% RSLogix 500 project 2 Head Filler - Reautomation.RSS, saved by version 7.00.00.19 %
PROJECT "ACINEW07"    % processor: MicroLogix 1200 %

PROGRAM FILES
  LAD 2 "MAIN"  15 rungs
  LAD 3 "FILL SEQ"  10 rungs
  LAD 4 "RESET"  12 rungs
  LAD 5 "HMI"  10 rungs
  LAD 6 "RECAP"  12 rungs

DATA FILES
  O0 OUTPUT  4 elements
  I1 INPUT  4 elements
  S2 STATUS  66 elements
  B3 BINARY  21 elements
  T4 TIMER  38 elements
  C5 COUNTER  1 elements
  R6 CONTROL  1 elements
  N7 INTEGER  7 elements
  F8 FLOAT  1 elements
  L9   1 elements

LADDER 2 "MAIN"
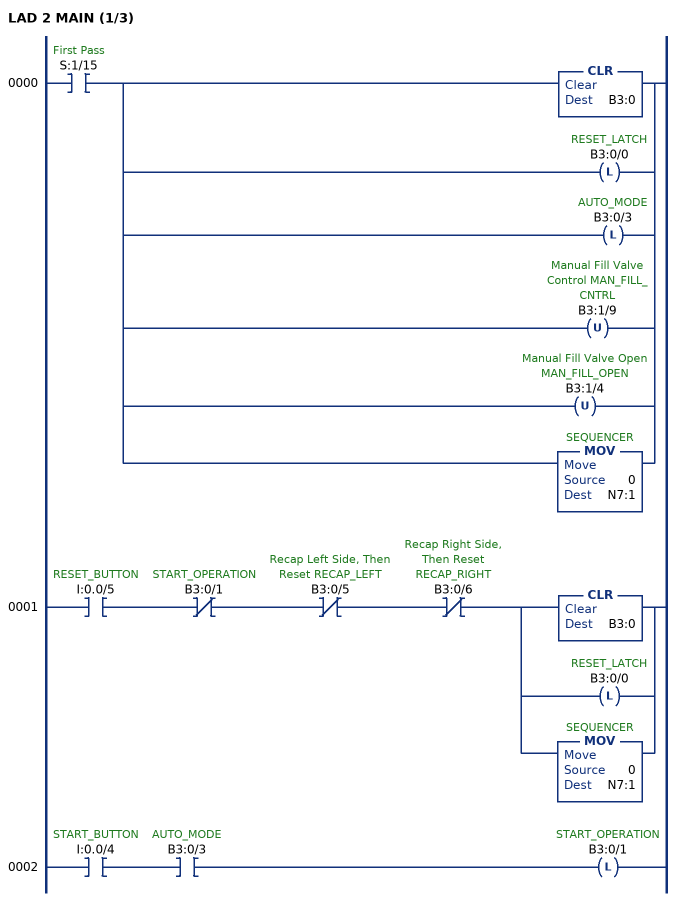
% Rung: 0 %
SOR XIC S:1/15 BST CLR B3:0 NXB OTL B3:0/0 NXB OTL B3:0/3 NXB OTU B3:1/9 NXB OTU B3:1/4 NXB MOV 0 N7:1 BND EOR
%   S:1/15  "First Pass" %
%   B3:0/0  RESET_LATCH %
%   B3:0/3  AUTO_MODE %
%   B3:1/9  MAN_FILL_CNTRL  "Manual Fill Valve Control" %
%   B3:1/4  MAN_FILL_OPEN  "Manual Fill Valve Open" %
%   N7:1  SEQUENCER %
% Rung: 1 %
SOR XIC I:0.0/5 XIO B3:0/1 XIO B3:0/5 XIO B3:0/6 BST CLR B3:0 NXB OTL B3:0/0 NXB MOV 0 N7:1 BND EOR
%   I:0.0/5  RESET_BUTTON %
%   B3:0/1  START_OPERATION %
%   B3:0/5  RECAP_LEFT  "Recap Left Side, Then Reset" %
%   B3:0/6  RECAP_RIGHT  "Recap Right Side, Then Reset" %
%   B3:0/0  RESET_LATCH %
%   N7:1  SEQUENCER %
% Rung: 2 %
SOR XIC I:0.0/4 XIC B3:0/3 OTL B3:0/1 EOR
%   I:0.0/4  START_BUTTON %
%   B3:0/3  AUTO_MODE %
%   B3:0/1  START_OPERATION %

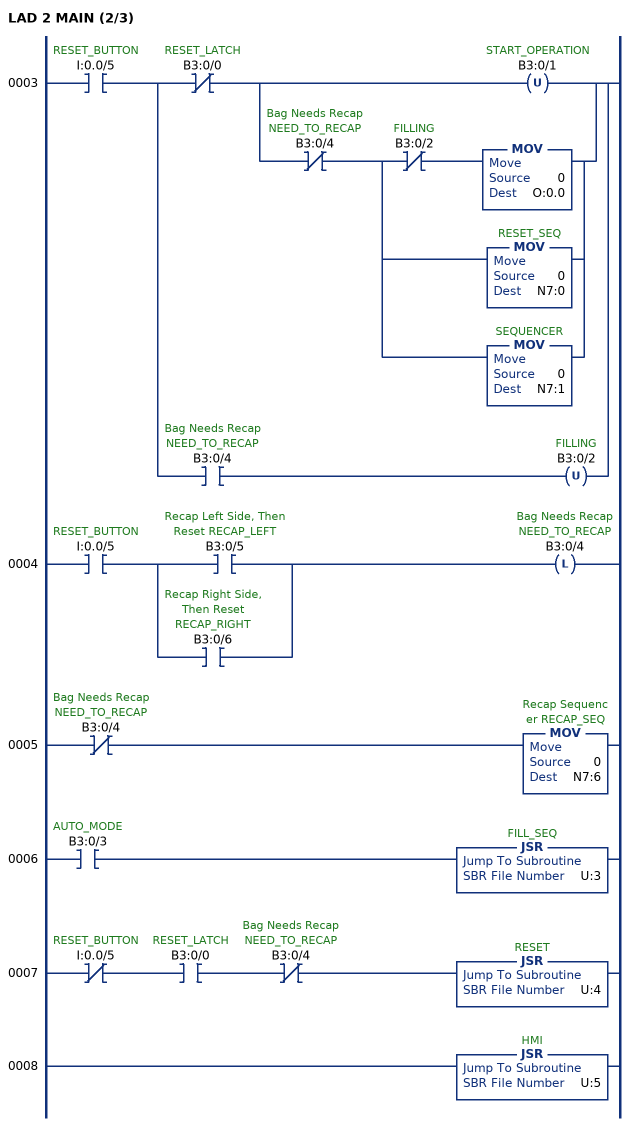
% Rung: 3 %
SOR XIC I:0.0/5 BST XIO B3:0/0 BST OTU B3:0/1 NXB XIO B3:0/4 BST XIO B3:0/2 MOV 0 O:0.0 NXB MOV 0 N7:0 NXB MOV 0 N7:1 BND BND NXB XIC B3:0/4 OTU B3:0/2 BND EOR
%   I:0.0/5  RESET_BUTTON %
%   B3:0/0  RESET_LATCH %
%   B3:0/1  START_OPERATION %
%   B3:0/4  NEED_TO_RECAP  "Bag Needs Recap" %
%   B3:0/2  FILLING %
%   N7:0  RESET_SEQ %
%   N7:1  SEQUENCER %
% Rung: 4 %
SOR XIC I:0.0/5 BST XIC B3:0/5 NXB XIC B3:0/6 BND OTL B3:0/4 EOR
%   I:0.0/5  RESET_BUTTON %
%   B3:0/5  RECAP_LEFT  "Recap Left Side, Then Reset" %
%   B3:0/6  RECAP_RIGHT  "Recap Right Side, Then Reset" %
%   B3:0/4  NEED_TO_RECAP  "Bag Needs Recap" %
% Rung: 5 %
SOR XIO B3:0/4 MOV 0 N7:6 EOR
%   B3:0/4  NEED_TO_RECAP  "Bag Needs Recap" %
%   N7:6  RECAP_SEQ  "Recap Sequencer" %
% Rung: 6 %
SOR XIC B3:0/3 JSR U:3 EOR
%   B3:0/3  AUTO_MODE %
%   U:3  FILL_SEQ %
% Rung: 7 %
SOR XIO I:0.0/5 XIC B3:0/0 XIO B3:0/4 JSR U:4 EOR
%   I:0.0/5  RESET_BUTTON %
%   B3:0/0  RESET_LATCH %
%   B3:0/4  NEED_TO_RECAP  "Bag Needs Recap" %
%   U:4  RESET %
% Rung: 8 %
SOR JSR U:5 EOR
%   U:5  HMI %

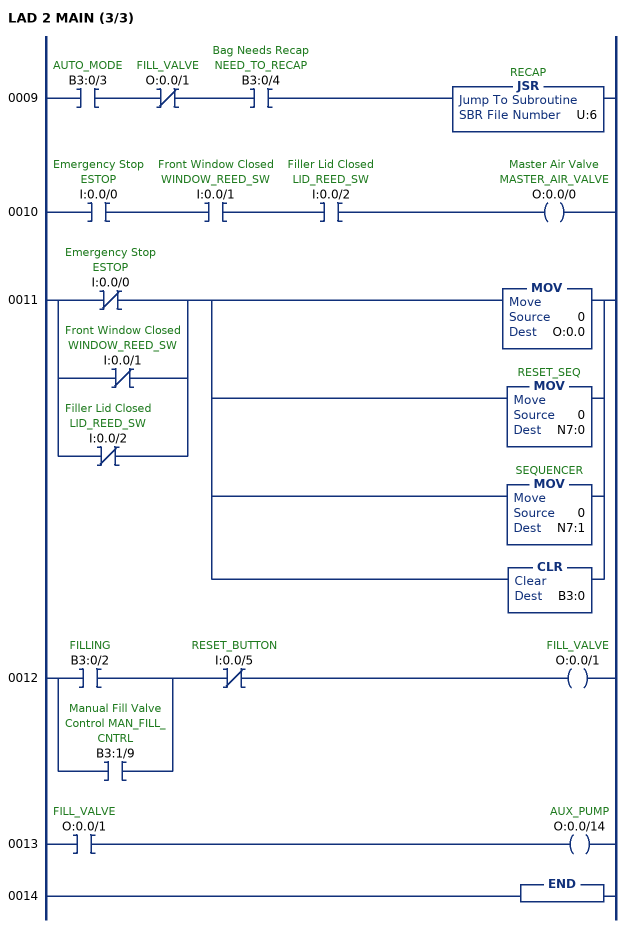
% Rung: 9 %
SOR XIC B3:0/3 XIO O:0.0/1 XIC B3:0/4 JSR U:6 EOR
%   B3:0/3  AUTO_MODE %
%   O:0.0/1  FILL_VALVE %
%   B3:0/4  NEED_TO_RECAP  "Bag Needs Recap" %
%   U:6  RECAP %
% Rung: 10 %
SOR XIC I:0.0/0 XIC I:0.0/1 XIC I:0.0/2 OTE O:0.0/0 EOR
%   I:0.0/0  ESTOP  "Emergency Stop" %
%   I:0.0/1  WINDOW_REED_SW  "Front Window Closed" %
%   I:0.0/2  LID_REED_SW  "Filler Lid Closed" %
%   O:0.0/0  MASTER_AIR_VALVE  "Master Air Valve" %
% Rung: 11 %
SOR BST XIO I:0.0/0 NXB XIO I:0.0/1 NXB XIO I:0.0/2 BND BST MOV 0 O:0.0 NXB MOV 0 N7:0 NXB MOV 0 N7:1 NXB CLR B3:0 BND EOR
%   I:0.0/0  ESTOP  "Emergency Stop" %
%   I:0.0/1  WINDOW_REED_SW  "Front Window Closed" %
%   I:0.0/2  LID_REED_SW  "Filler Lid Closed" %
%   N7:0  RESET_SEQ %
%   N7:1  SEQUENCER %
% Rung: 12 %
SOR BST XIC B3:0/2 NXB XIC B3:1/9 BND XIO I:0.0/5 OTE O:0.0/1 EOR
%   B3:0/2  FILLING %
%   B3:1/9  MAN_FILL_CNTRL  "Manual Fill Valve Control" %
%   I:0.0/5  RESET_BUTTON %
%   O:0.0/1  FILL_VALVE %
% Rung: 13 %
SOR XIC O:0.0/1 OTE O:0.0/14 EOR
%   O:0.0/1  FILL_VALVE %
%   O:0.0/14  AUX_PUMP %
% Rung: 14 %
SOR END EOR

LADDER 3 "FILL SEQ"
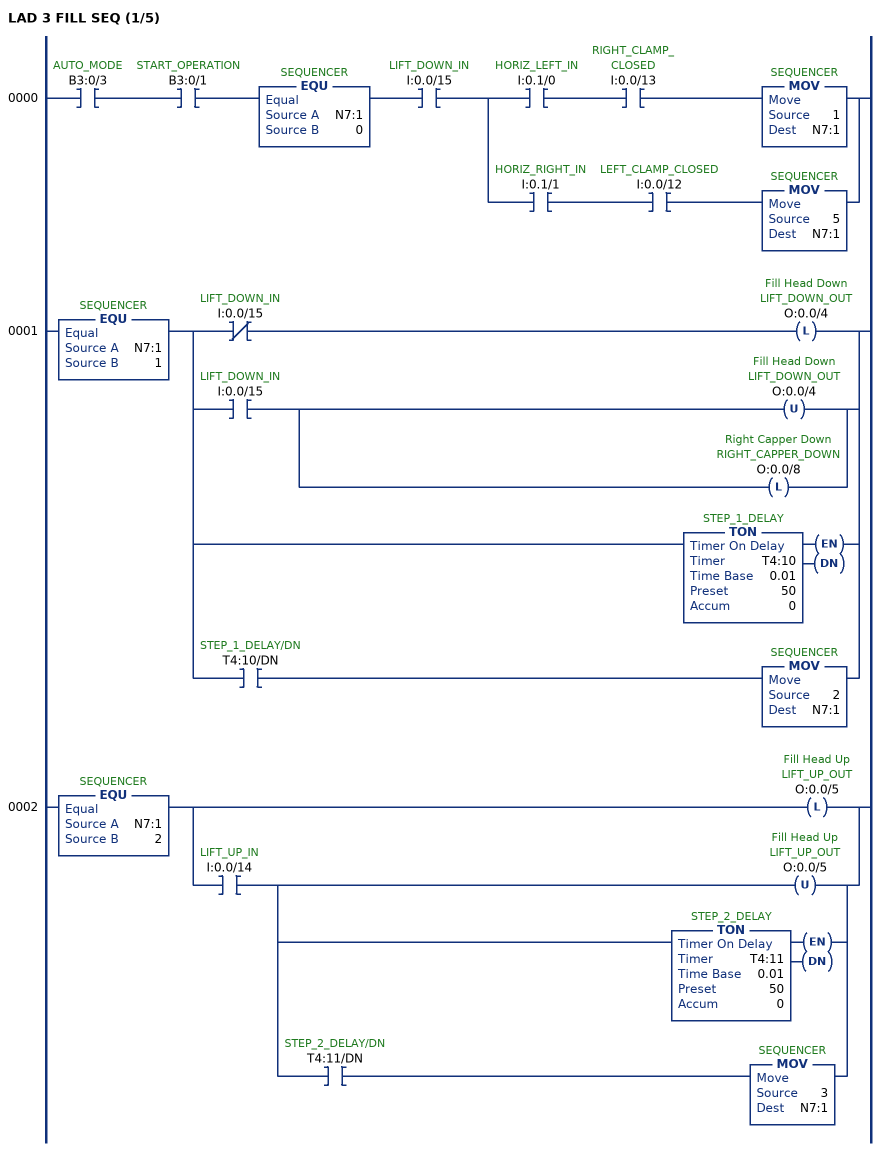
% Rung: 0 %
SOR XIC B3:0/3 XIC B3:0/1 EQU N7:1 0 XIC I:0.0/15 BST XIC I:0.1/0 XIC I:0.0/13 MOV 1 N7:1 NXB XIC I:0.1/1 XIC I:0.0/12 MOV 5 N7:1 BND EOR
%   B3:0/3  AUTO_MODE %
%   B3:0/1  START_OPERATION %
%   N7:1  SEQUENCER %
%   I:0.0/15  LIFT_DOWN_IN %
%   I:0.1/0  HORIZ_LEFT_IN %
%   I:0.0/13  RIGHT_CLAMP_CLOSED %
%   I:0.1/1  HORIZ_RIGHT_IN %
%   I:0.0/12  LEFT_CLAMP_CLOSED %
% Rung: 1 %
SOR EQU N7:1 1 BST XIO I:0.0/15 OTL O:0.0/4 NXB XIC I:0.0/15 BST OTU O:0.0/4 NXB OTL O:0.0/8 BND NXB TON T4:10 0.01 50 0 NXB XIC T4:10/DN MOV 2 N7:1 BND EOR
%   N7:1  SEQUENCER %
%   I:0.0/15  LIFT_DOWN_IN %
%   O:0.0/4  LIFT_DOWN_OUT  "Fill Head Down" %
%   O:0.0/8  RIGHT_CAPPER_DOWN  "Right Capper Down" %
%   T4:10  STEP_1_DELAY %
% Rung: 2 %
SOR EQU N7:1 2 BST OTL O:0.0/5 NXB XIC I:0.0/14 BST OTU O:0.0/5 NXB TON T4:11 0.01 50 0 NXB XIC T4:11/DN MOV 3 N7:1 BND BND EOR
%   N7:1  SEQUENCER %
%   O:0.0/5  LIFT_UP_OUT  "Fill Head Up" %
%   I:0.0/14  LIFT_UP_IN %
%   T4:11  STEP_2_DELAY %

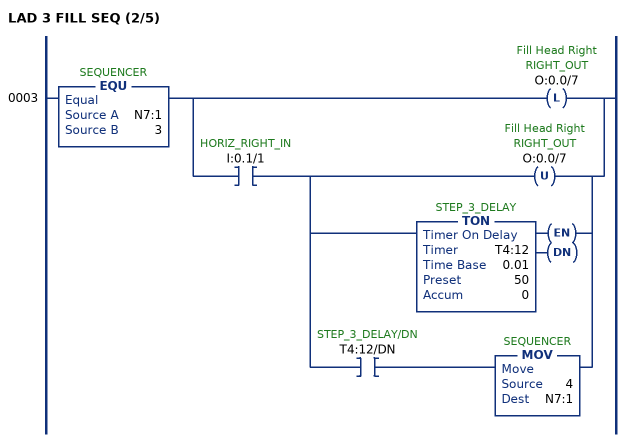
% Rung: 3 %
SOR EQU N7:1 3 BST OTL O:0.0/7 NXB XIC I:0.1/1 BST OTU O:0.0/7 NXB TON T4:12 0.01 50 0 NXB XIC T4:12/DN MOV 4 N7:1 BND BND EOR
%   N7:1  SEQUENCER %
%   O:0.0/7  RIGHT_OUT  "Fill Head Right" %
%   I:0.1/1  HORIZ_RIGHT_IN %
%   T4:12  STEP_3_DELAY %

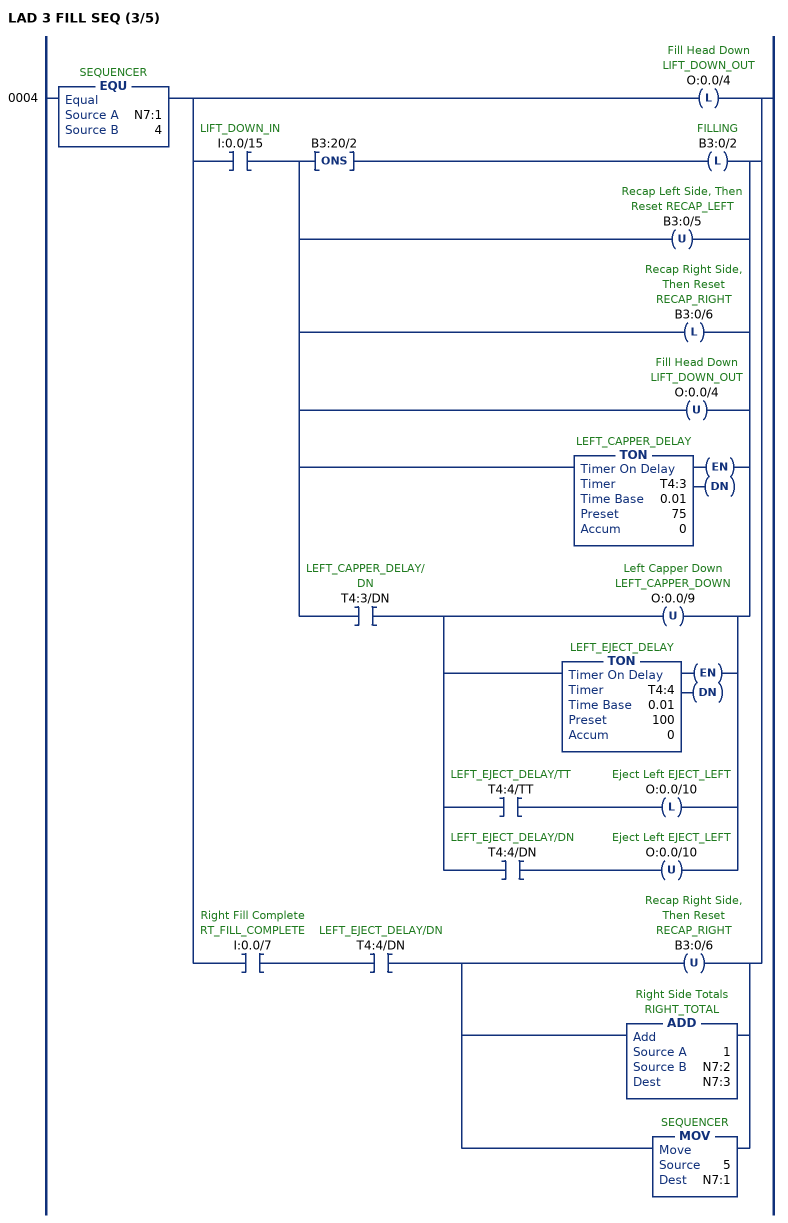
% Rung: 4 %
SOR EQU N7:1 4 BST OTL O:0.0/4 NXB XIC I:0.0/15 BST ONS B3:20/2 OTL B3:0/2 NXB OTU B3:0/5 NXB OTL B3:0/6 NXB OTU O:0.0/4 NXB TON T4:3 0.01 75 0 NXB XIC T4:3/DN BST OTU O:0.0/9 NXB TON T4:4 0.01 100 0 NXB XIC T4:4/TT OTL O:0.0/10 NXB XIC T4:4/DN OTU O:0.0/10 BND BND NXB XIC I:0.0/7 XIC T4:4/DN BST OTU B3:0/6 NXB ADD 1 N7:2 N7:3 NXB MOV 5 N7:1 BND BND EOR
%   N7:1  SEQUENCER %
%   O:0.0/4  LIFT_DOWN_OUT  "Fill Head Down" %
%   I:0.0/15  LIFT_DOWN_IN %
%   B3:0/2  FILLING %
%   B3:0/5  RECAP_LEFT  "Recap Left Side, Then Reset" %
%   B3:0/6  RECAP_RIGHT  "Recap Right Side, Then Reset" %
%   T4:3  LEFT_CAPPER_DELAY %
%   O:0.0/9  LEFT_CAPPER_DOWN  "Left Capper Down" %
%   T4:4  LEFT_EJECT_DELAY %
%   O:0.0/10  EJECT_LEFT  "Eject Left" %
%   I:0.0/7  RT_FILL_COMPLETE  "Right Fill Complete" %
%   N7:2  LEFT_TOTAL  "Left Side Totals" %
%   N7:3  RIGHT_TOTAL  "Right Side Totals" %

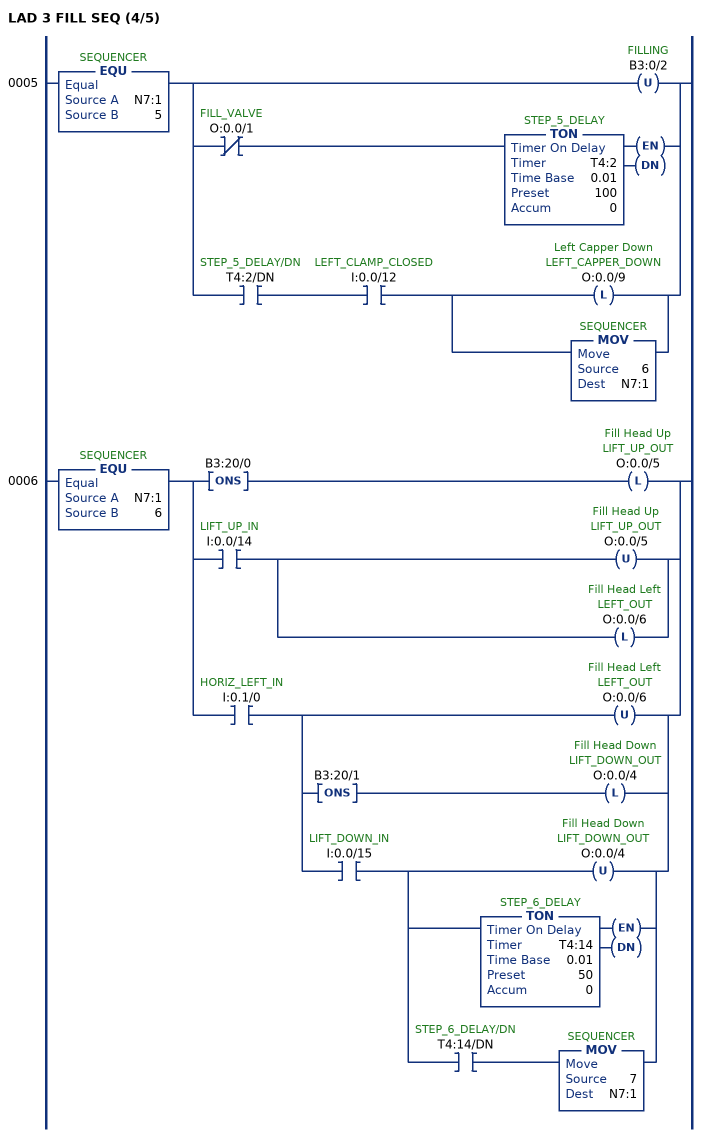
% Rung: 5 %
SOR EQU N7:1 5 BST OTU B3:0/2 NXB XIO O:0.0/1 TON T4:2 0.01 100 0 NXB XIC T4:2/DN XIC I:0.0/12 BST OTL O:0.0/9 NXB MOV 6 N7:1 BND BND EOR
%   N7:1  SEQUENCER %
%   B3:0/2  FILLING %
%   O:0.0/1  FILL_VALVE %
%   T4:2  STEP_5_DELAY %
%   I:0.0/12  LEFT_CLAMP_CLOSED %
%   O:0.0/9  LEFT_CAPPER_DOWN  "Left Capper Down" %
% Rung: 6 %
SOR EQU N7:1 6 BST ONS B3:20/0 OTL O:0.0/5 NXB BST XIC I:0.0/14 BST OTU O:0.0/5 NXB OTL O:0.0/6 BND NXB XIC I:0.1/0 BST OTU O:0.0/6 NXB ONS B3:20/1 OTL O:0.0/4 NXB XIC I:0.0/15 BST OTU O:0.0/4 NXB TON T4:14 0.01 50 0 NXB XIC T4:14/DN MOV 7 N7:1 BND BND BND BND EOR
%   N7:1  SEQUENCER %
%   O:0.0/5  LIFT_UP_OUT  "Fill Head Up" %
%   I:0.0/14  LIFT_UP_IN %
%   O:0.0/6  LEFT_OUT  "Fill Head Left" %
%   I:0.1/0  HORIZ_LEFT_IN %
%   O:0.0/4  LIFT_DOWN_OUT  "Fill Head Down" %
%   I:0.0/15  LIFT_DOWN_IN %
%   T4:14  STEP_6_DELAY %

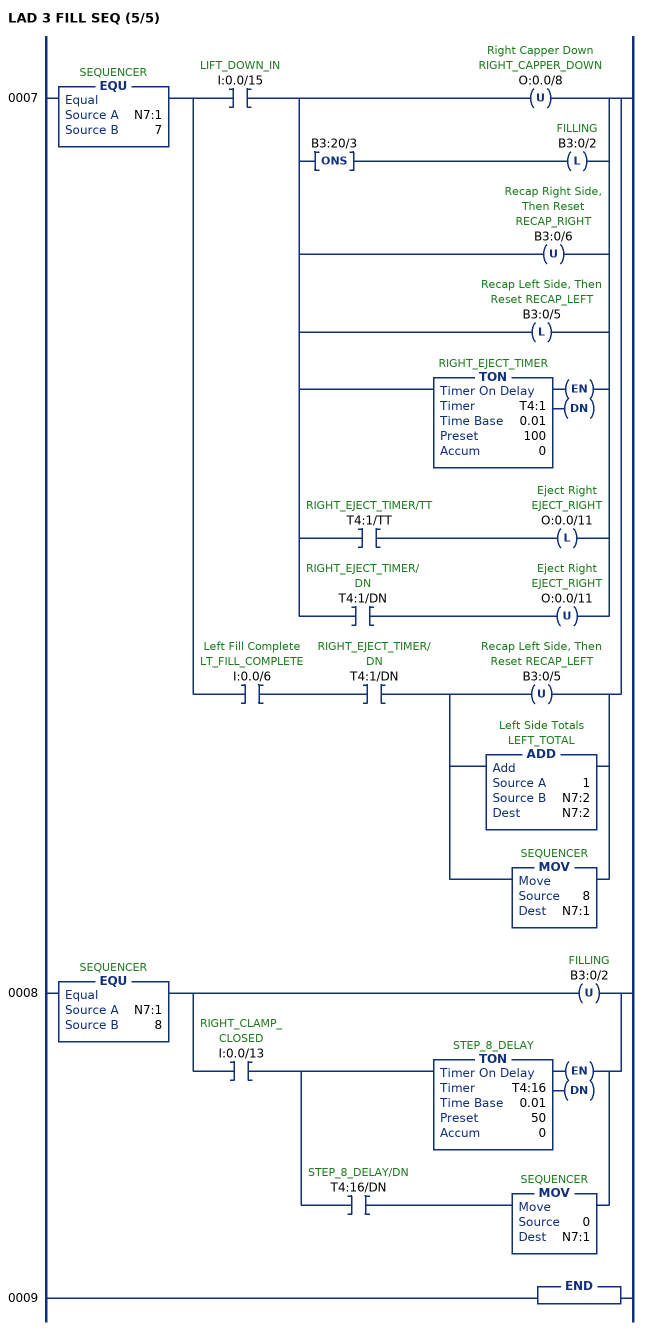
% Rung: 7 %
SOR EQU N7:1 7 BST XIC I:0.0/15 BST OTU O:0.0/8 NXB ONS B3:20/3 OTL B3:0/2 NXB OTU B3:0/6 NXB OTL B3:0/5 NXB TON T4:1 0.01 100 0 NXB XIC T4:1/TT OTL O:0.0/11 NXB XIC T4:1/DN OTU O:0.0/11 BND NXB XIC I:0.0/6 XIC T4:1/DN BST OTU B3:0/5 NXB ADD 1 N7:2 N7:2 NXB MOV 8 N7:1 BND BND EOR
%   N7:1  SEQUENCER %
%   I:0.0/15  LIFT_DOWN_IN %
%   O:0.0/8  RIGHT_CAPPER_DOWN  "Right Capper Down" %
%   B3:0/2  FILLING %
%   B3:0/6  RECAP_RIGHT  "Recap Right Side, Then Reset" %
%   B3:0/5  RECAP_LEFT  "Recap Left Side, Then Reset" %
%   T4:1  RIGHT_EJECT_TIMER %
%   O:0.0/11  EJECT_RIGHT  "Eject Right" %
%   I:0.0/6  LT_FILL_COMPLETE  "Left Fill Complete" %
%   N7:2  LEFT_TOTAL  "Left Side Totals" %
% Rung: 8 %
SOR EQU N7:1 8 BST OTU B3:0/2 NXB XIC I:0.0/13 BST TON T4:16 0.01 50 0 NXB XIC T4:16/DN MOV 0 N7:1 BND BND EOR
%   N7:1  SEQUENCER %
%   B3:0/2  FILLING %
%   I:0.0/13  RIGHT_CLAMP_CLOSED %
%   T4:16  STEP_8_DELAY %
% Rung: 9 %
SOR END EOR

LADDER 4 "RESET"
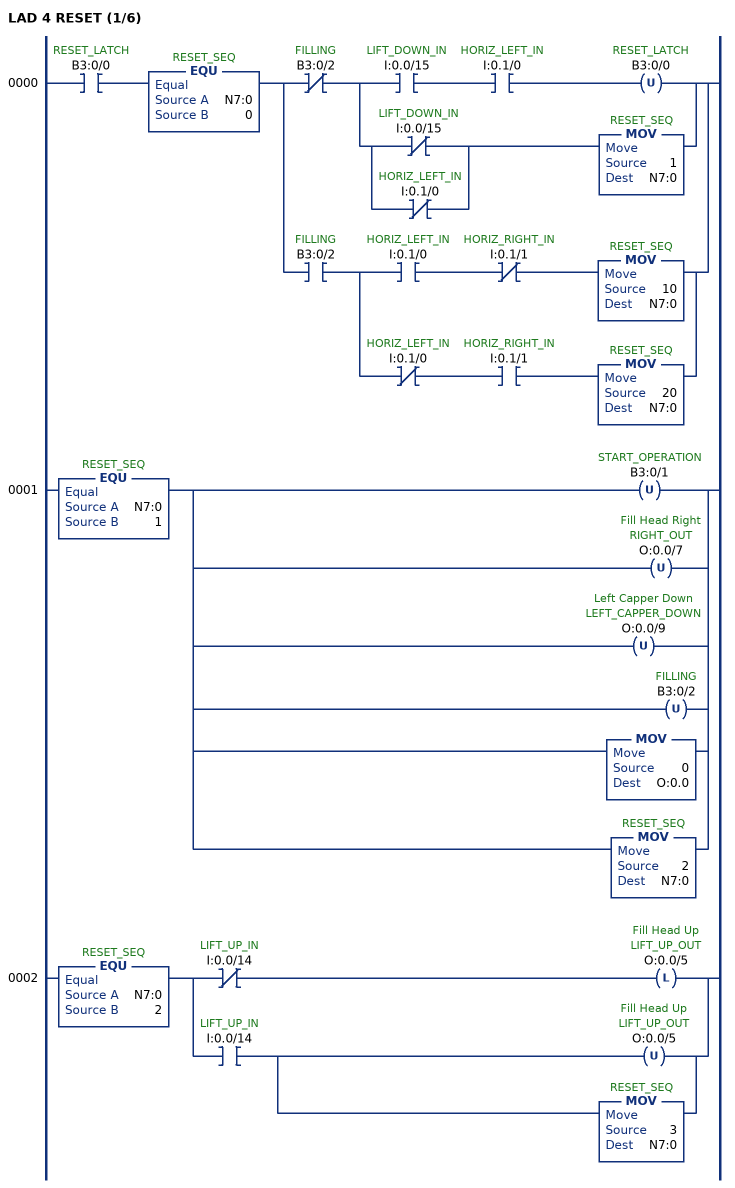
% Rung: 0 %
SOR XIC B3:0/0 EQU N7:0 0 BST XIO B3:0/2 BST XIC I:0.0/15 XIC I:0.1/0 OTU B3:0/0 NXB BST XIO I:0.0/15 NXB XIO I:0.1/0 BND MOV 1 N7:0 BND NXB XIC B3:0/2 BST XIC I:0.1/0 XIO I:0.1/1 MOV 10 N7:0 NXB XIO I:0.1/0 XIC I:0.1/1 MOV 20 N7:0 BND BND EOR
%   B3:0/0  RESET_LATCH %
%   N7:0  RESET_SEQ %
%   B3:0/2  FILLING %
%   I:0.0/15  LIFT_DOWN_IN %
%   I:0.1/0  HORIZ_LEFT_IN %
%   I:0.1/1  HORIZ_RIGHT_IN %
% Rung: 1 %
SOR EQU N7:0 1 BST OTU B3:0/1 NXB OTU O:0.0/7 NXB OTU O:0.0/9 NXB OTU B3:0/2 NXB MOV 0 O:0.0 NXB MOV 2 N7:0 BND EOR
%   N7:0  RESET_SEQ %
%   B3:0/1  START_OPERATION %
%   O:0.0/7  RIGHT_OUT  "Fill Head Right" %
%   O:0.0/9  LEFT_CAPPER_DOWN  "Left Capper Down" %
%   B3:0/2  FILLING %
% Rung: 2 %
SOR EQU N7:0 2 BST XIO I:0.0/14 OTL O:0.0/5 NXB XIC I:0.0/14 BST OTU O:0.0/5 NXB MOV 3 N7:0 BND BND EOR
%   N7:0  RESET_SEQ %
%   I:0.0/14  LIFT_UP_IN %
%   O:0.0/5  LIFT_UP_OUT  "Fill Head Up" %

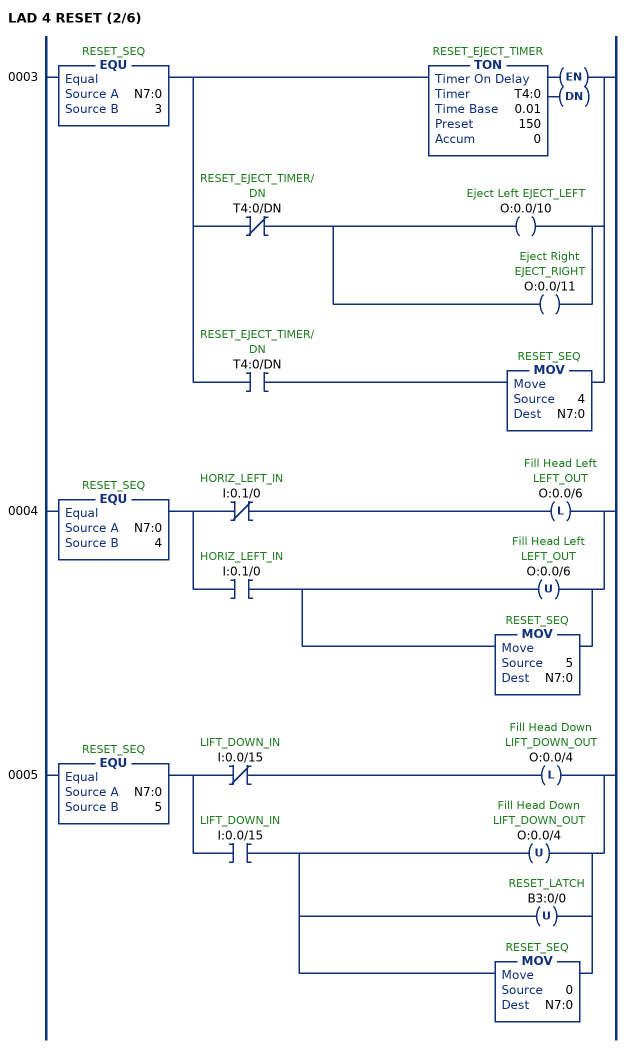
% Rung: 3 %
SOR EQU N7:0 3 BST TON T4:0 0.01 150 0 NXB XIO T4:0/DN BST OTE O:0.0/10 NXB OTE O:0.0/11 BND NXB XIC T4:0/DN MOV 4 N7:0 BND EOR
%   N7:0  RESET_SEQ %
%   T4:0  RESET_EJECT_TIMER %
%   O:0.0/10  EJECT_LEFT  "Eject Left" %
%   O:0.0/11  EJECT_RIGHT  "Eject Right" %
% Rung: 4 %
SOR EQU N7:0 4 BST XIO I:0.1/0 OTL O:0.0/6 NXB XIC I:0.1/0 BST OTU O:0.0/6 NXB MOV 5 N7:0 BND BND EOR
%   N7:0  RESET_SEQ %
%   I:0.1/0  HORIZ_LEFT_IN %
%   O:0.0/6  LEFT_OUT  "Fill Head Left" %
% Rung: 5 %
SOR EQU N7:0 5 BST XIO I:0.0/15 OTL O:0.0/4 NXB XIC I:0.0/15 BST OTU O:0.0/4 NXB OTU B3:0/0 NXB MOV 0 N7:0 BND BND EOR
%   N7:0  RESET_SEQ %
%   I:0.0/15  LIFT_DOWN_IN %
%   O:0.0/4  LIFT_DOWN_OUT  "Fill Head Down" %
%   B3:0/0  RESET_LATCH %

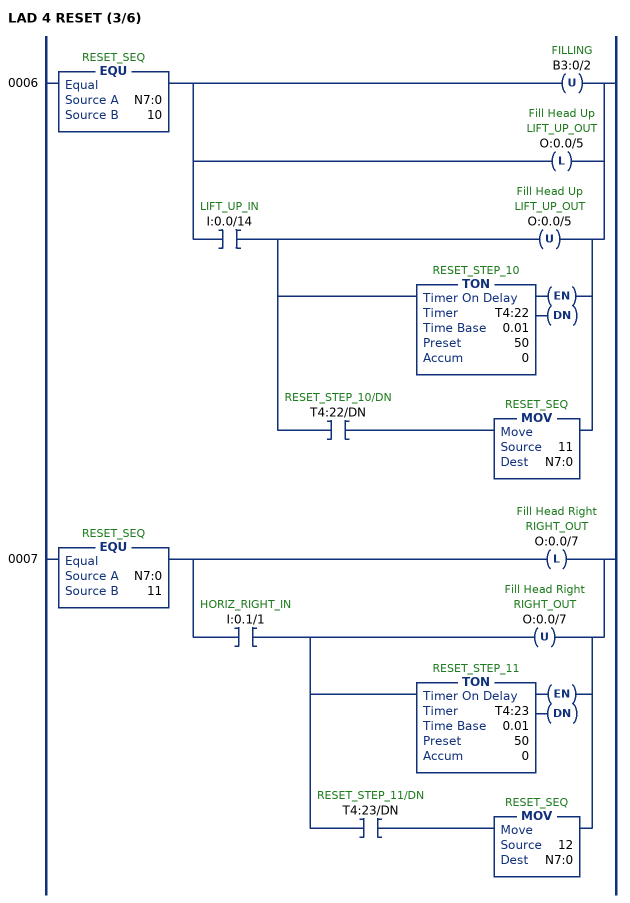
% Rung: 6 %
SOR EQU N7:0 10 BST OTU B3:0/2 NXB OTL O:0.0/5 NXB XIC I:0.0/14 BST OTU O:0.0/5 NXB TON T4:22 0.01 50 0 NXB XIC T4:22/DN MOV 11 N7:0 BND BND EOR
%   N7:0  RESET_SEQ %
%   B3:0/2  FILLING %
%   O:0.0/5  LIFT_UP_OUT  "Fill Head Up" %
%   I:0.0/14  LIFT_UP_IN %
%   T4:22  RESET_STEP_10 %
% Rung: 7 %
SOR EQU N7:0 11 BST OTL O:0.0/7 NXB XIC I:0.1/1 BST OTU O:0.0/7 NXB TON T4:23 0.01 50 0 NXB XIC T4:23/DN MOV 12 N7:0 BND BND EOR
%   N7:0  RESET_SEQ %
%   O:0.0/7  RIGHT_OUT  "Fill Head Right" %
%   I:0.1/1  HORIZ_RIGHT_IN %
%   T4:23  RESET_STEP_11 %

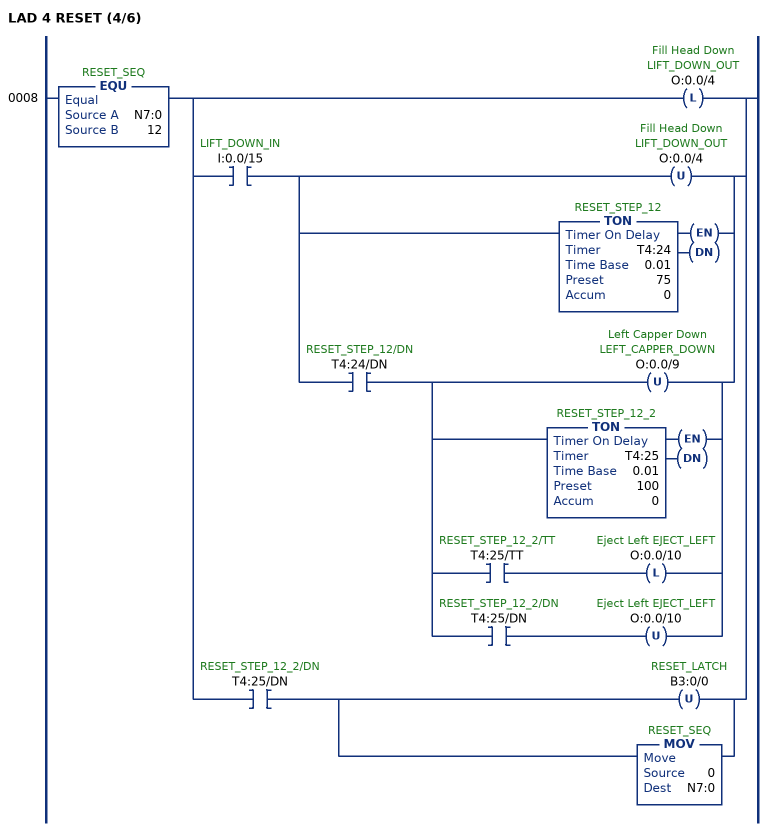
% Rung: 8 %
SOR EQU N7:0 12 BST OTL O:0.0/4 NXB XIC I:0.0/15 BST OTU O:0.0/4 NXB TON T4:24 0.01 75 0 NXB XIC T4:24/DN BST OTU O:0.0/9 NXB TON T4:25 0.01 100 0 NXB XIC T4:25/TT OTL O:0.0/10 NXB XIC T4:25/DN OTU O:0.0/10 BND BND NXB XIC T4:25/DN BST OTU B3:0/0 NXB MOV 0 N7:0 BND BND EOR
%   N7:0  RESET_SEQ %
%   O:0.0/4  LIFT_DOWN_OUT  "Fill Head Down" %
%   I:0.0/15  LIFT_DOWN_IN %
%   T4:24  RESET_STEP_12 %
%   O:0.0/9  LEFT_CAPPER_DOWN  "Left Capper Down" %
%   T4:25  RESET_STEP_12_2 %
%   O:0.0/10  EJECT_LEFT  "Eject Left" %
%   B3:0/0  RESET_LATCH %

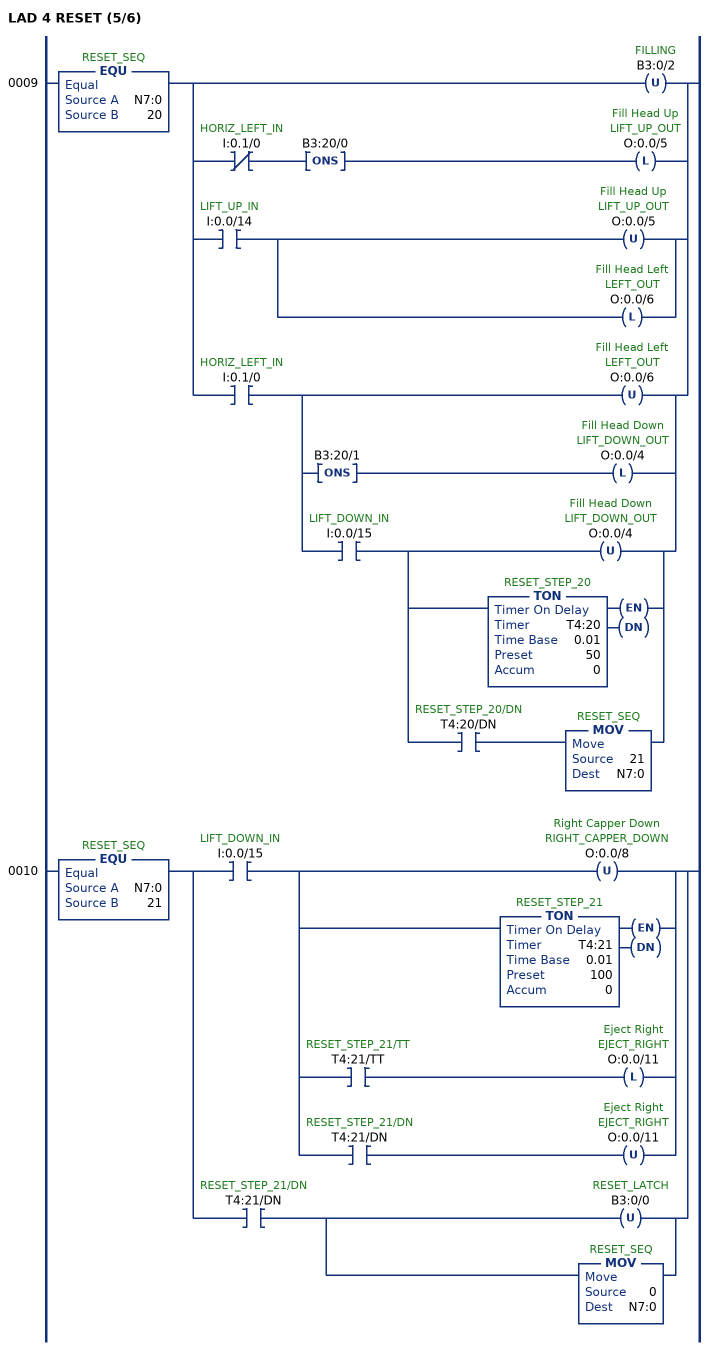
% Rung: 9 %
SOR EQU N7:0 20 BST OTU B3:0/2 NXB XIO I:0.1/0 ONS B3:20/0 OTL O:0.0/5 NXB BST XIC I:0.0/14 BST OTU O:0.0/5 NXB OTL O:0.0/6 BND NXB XIC I:0.1/0 BST OTU O:0.0/6 NXB ONS B3:20/1 OTL O:0.0/4 NXB XIC I:0.0/15 BST OTU O:0.0/4 NXB TON T4:20 0.01 50 0 NXB XIC T4:20/DN MOV 21 N7:0 BND BND BND BND EOR
%   N7:0  RESET_SEQ %
%   B3:0/2  FILLING %
%   I:0.1/0  HORIZ_LEFT_IN %
%   O:0.0/5  LIFT_UP_OUT  "Fill Head Up" %
%   I:0.0/14  LIFT_UP_IN %
%   O:0.0/6  LEFT_OUT  "Fill Head Left" %
%   O:0.0/4  LIFT_DOWN_OUT  "Fill Head Down" %
%   I:0.0/15  LIFT_DOWN_IN %
%   T4:20  RESET_STEP_20 %
% Rung: 10 %
SOR EQU N7:0 21 BST XIC I:0.0/15 BST OTU O:0.0/8 NXB TON T4:21 0.01 100 0 NXB XIC T4:21/TT OTL O:0.0/11 NXB XIC T4:21/DN OTU O:0.0/11 BND NXB XIC T4:21/DN BST OTU B3:0/0 NXB MOV 0 N7:0 BND BND EOR
%   N7:0  RESET_SEQ %
%   I:0.0/15  LIFT_DOWN_IN %
%   O:0.0/8  RIGHT_CAPPER_DOWN  "Right Capper Down" %
%   T4:21  RESET_STEP_21 %
%   O:0.0/11  EJECT_RIGHT  "Eject Right" %
%   B3:0/0  RESET_LATCH %

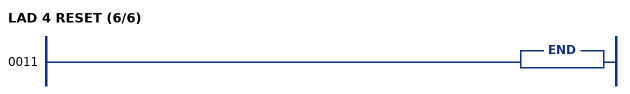
% Rung: 11 %
SOR END EOR

LADDER 5 "HMI"
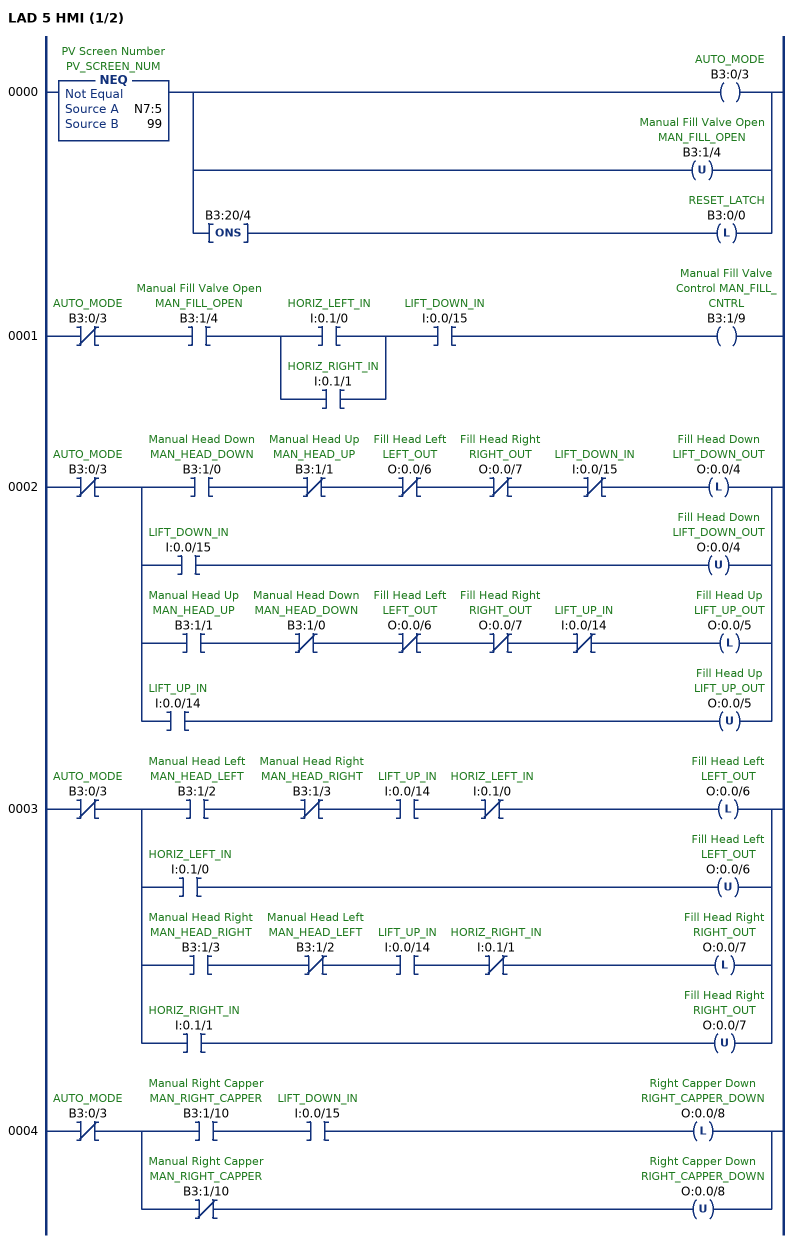
% Rung: 0 %
SOR NEQ N7:5 99 BST OTE B3:0/3 NXB OTU B3:1/4 NXB ONS B3:20/4 OTL B3:0/0 BND EOR
%   N7:5  PV_SCREEN_NUM  "PV Screen Number" %
%   B3:0/3  AUTO_MODE %
%   B3:1/4  MAN_FILL_OPEN  "Manual Fill Valve Open" %
%   B3:0/0  RESET_LATCH %
% Rung: 1 %
SOR XIO B3:0/3 XIC B3:1/4 BST XIC I:0.1/0 NXB XIC I:0.1/1 BND XIC I:0.0/15 OTE B3:1/9 EOR
%   B3:0/3  AUTO_MODE %
%   B3:1/4  MAN_FILL_OPEN  "Manual Fill Valve Open" %
%   I:0.1/0  HORIZ_LEFT_IN %
%   I:0.1/1  HORIZ_RIGHT_IN %
%   I:0.0/15  LIFT_DOWN_IN %
%   B3:1/9  MAN_FILL_CNTRL  "Manual Fill Valve Control" %
% Rung: 2 %
SOR XIO B3:0/3 BST XIC B3:1/0 XIO B3:1/1 XIO O:0.0/6 XIO O:0.0/7 XIO I:0.0/15 OTL O:0.0/4 NXB XIC I:0.0/15 OTU O:0.0/4 NXB XIC B3:1/1 XIO B3:1/0 XIO O:0.0/6 XIO O:0.0/7 XIO I:0.0/14 OTL O:0.0/5 NXB XIC I:0.0/14 OTU O:0.0/5 BND EOR
%   B3:0/3  AUTO_MODE %
%   B3:1/0  MAN_HEAD_DOWN  "Manual Head Down" %
%   B3:1/1  MAN_HEAD_UP  "Manual Head Up" %
%   O:0.0/6  LEFT_OUT  "Fill Head Left" %
%   O:0.0/7  RIGHT_OUT  "Fill Head Right" %
%   I:0.0/15  LIFT_DOWN_IN %
%   O:0.0/4  LIFT_DOWN_OUT  "Fill Head Down" %
%   I:0.0/14  LIFT_UP_IN %
%   O:0.0/5  LIFT_UP_OUT  "Fill Head Up" %
% Rung: 3 %
SOR XIO B3:0/3 BST XIC B3:1/2 XIO B3:1/3 XIC I:0.0/14 XIO I:0.1/0 OTL O:0.0/6 NXB XIC I:0.1/0 OTU O:0.0/6 NXB XIC B3:1/3 XIO B3:1/2 XIC I:0.0/14 XIO I:0.1/1 OTL O:0.0/7 NXB XIC I:0.1/1 OTU O:0.0/7 BND EOR
%   B3:0/3  AUTO_MODE %
%   B3:1/2  MAN_HEAD_LEFT  "Manual Head Left" %
%   B3:1/3  MAN_HEAD_RIGHT  "Manual Head Right" %
%   I:0.0/14  LIFT_UP_IN %
%   I:0.1/0  HORIZ_LEFT_IN %
%   O:0.0/6  LEFT_OUT  "Fill Head Left" %
%   I:0.1/1  HORIZ_RIGHT_IN %
%   O:0.0/7  RIGHT_OUT  "Fill Head Right" %
% Rung: 4 %
SOR XIO B3:0/3 BST XIC B3:1/10 XIC I:0.0/15 OTL O:0.0/8 NXB XIO B3:1/10 OTU O:0.0/8 BND EOR
%   B3:0/3  AUTO_MODE %
%   B3:1/10  MAN_RIGHT_CAPPER  "Manual Right Capper" %
%   I:0.0/15  LIFT_DOWN_IN %
%   O:0.0/8  RIGHT_CAPPER_DOWN  "Right Capper Down" %

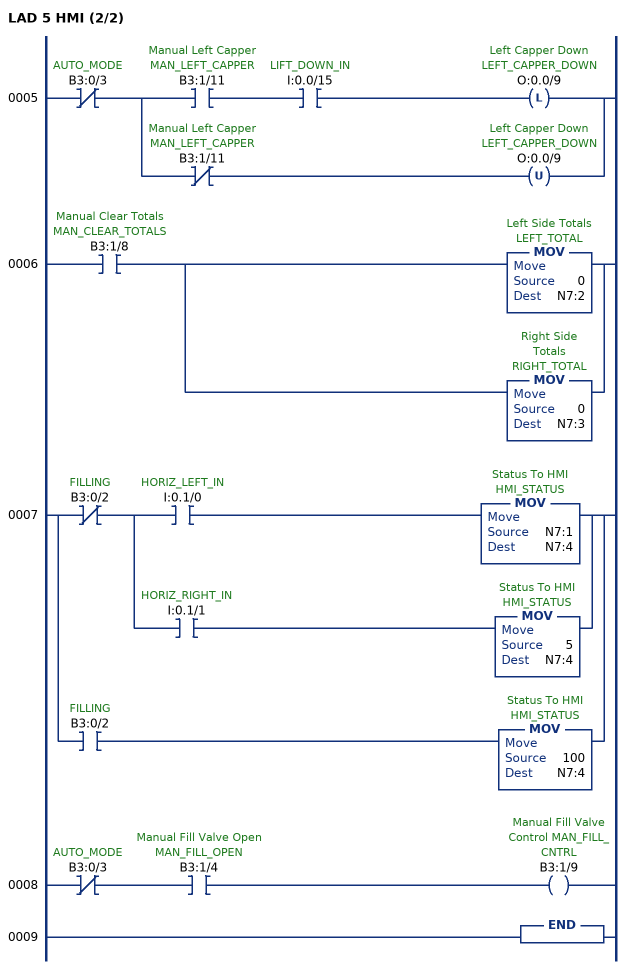
% Rung: 5 %
SOR XIO B3:0/3 BST XIC B3:1/11 XIC I:0.0/15 OTL O:0.0/9 NXB XIO B3:1/11 OTU O:0.0/9 BND EOR
%   B3:0/3  AUTO_MODE %
%   B3:1/11  MAN_LEFT_CAPPER  "Manual Left Capper" %
%   I:0.0/15  LIFT_DOWN_IN %
%   O:0.0/9  LEFT_CAPPER_DOWN  "Left Capper Down" %
% Rung: 6 %
SOR XIC B3:1/8 BST MOV 0 N7:2 NXB MOV 0 N7:3 BND EOR
%   B3:1/8  MAN_CLEAR_TOTALS  "Manual Clear Totals" %
%   N7:2  LEFT_TOTAL  "Left Side Totals" %
%   N7:3  RIGHT_TOTAL  "Right Side Totals" %
% Rung: 7 %
SOR BST XIO B3:0/2 BST XIC I:0.1/0 MOV N7:1 N7:4 NXB XIC I:0.1/1 MOV 5 N7:4 BND NXB XIC B3:0/2 MOV 100 N7:4 BND EOR
%   B3:0/2  FILLING %
%   I:0.1/0  HORIZ_LEFT_IN %
%   N7:1  SEQUENCER %
%   N7:4  HMI_STATUS  "Status To HMI" %
%   I:0.1/1  HORIZ_RIGHT_IN %
% Rung: 8 %
SOR XIO B3:0/3 XIC B3:1/4 OTE B3:1/9 EOR
%   B3:0/3  AUTO_MODE %
%   B3:1/4  MAN_FILL_OPEN  "Manual Fill Valve Open" %
%   B3:1/9  MAN_FILL_CNTRL  "Manual Fill Valve Control" %
% Rung: 9 %
SOR END EOR

LADDER 6 "RECAP"
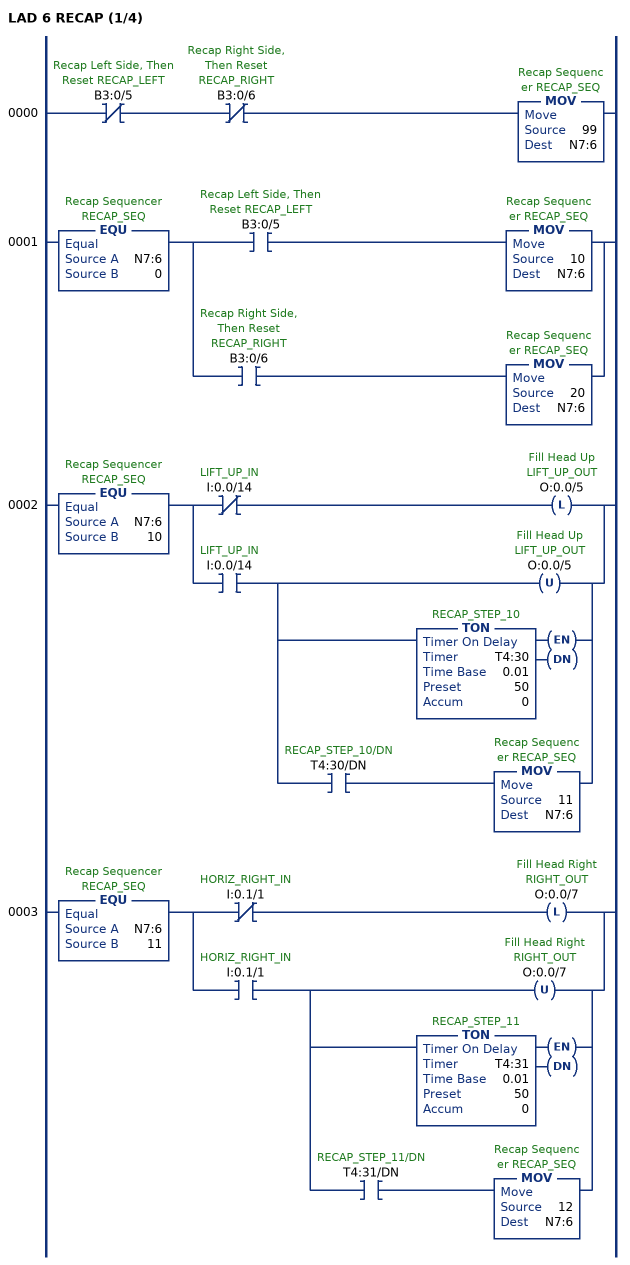
% Rung: 0 %
SOR XIO B3:0/5 XIO B3:0/6 MOV 99 N7:6 EOR
%   B3:0/5  RECAP_LEFT  "Recap Left Side, Then Reset" %
%   B3:0/6  RECAP_RIGHT  "Recap Right Side, Then Reset" %
%   N7:6  RECAP_SEQ  "Recap Sequencer" %
% Rung: 1 %
SOR EQU N7:6 0 BST XIC B3:0/5 MOV 10 N7:6 NXB XIC B3:0/6 MOV 20 N7:6 BND EOR
%   N7:6  RECAP_SEQ  "Recap Sequencer" %
%   B3:0/5  RECAP_LEFT  "Recap Left Side, Then Reset" %
%   B3:0/6  RECAP_RIGHT  "Recap Right Side, Then Reset" %
% Rung: 2 %
SOR EQU N7:6 10 BST XIO I:0.0/14 OTL O:0.0/5 NXB XIC I:0.0/14 BST OTU O:0.0/5 NXB TON T4:30 0.01 50 0 NXB XIC T4:30/DN MOV 11 N7:6 BND BND EOR
%   N7:6  RECAP_SEQ  "Recap Sequencer" %
%   I:0.0/14  LIFT_UP_IN %
%   O:0.0/5  LIFT_UP_OUT  "Fill Head Up" %
%   T4:30  RECAP_STEP_10 %
% Rung: 3 %
SOR EQU N7:6 11 BST XIO I:0.1/1 OTL O:0.0/7 NXB XIC I:0.1/1 BST OTU O:0.0/7 NXB TON T4:31 0.01 50 0 NXB XIC T4:31/DN MOV 12 N7:6 BND BND EOR
%   N7:6  RECAP_SEQ  "Recap Sequencer" %
%   I:0.1/1  HORIZ_RIGHT_IN %
%   O:0.0/7  RIGHT_OUT  "Fill Head Right" %
%   T4:31  RECAP_STEP_11 %

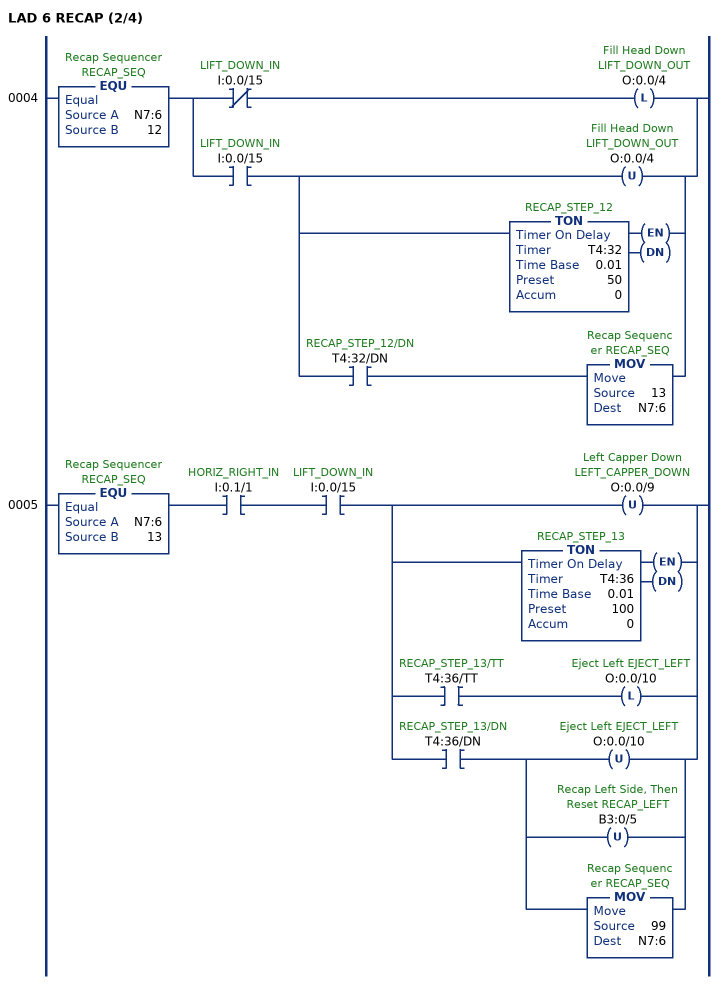
% Rung: 4 %
SOR EQU N7:6 12 BST XIO I:0.0/15 OTL O:0.0/4 NXB XIC I:0.0/15 BST OTU O:0.0/4 NXB TON T4:32 0.01 50 0 NXB XIC T4:32/DN MOV 13 N7:6 BND BND EOR
%   N7:6  RECAP_SEQ  "Recap Sequencer" %
%   I:0.0/15  LIFT_DOWN_IN %
%   O:0.0/4  LIFT_DOWN_OUT  "Fill Head Down" %
%   T4:32  RECAP_STEP_12 %
% Rung: 5 %
SOR EQU N7:6 13 XIC I:0.1/1 XIC I:0.0/15 BST OTU O:0.0/9 NXB TON T4:36 0.01 100 0 NXB XIC T4:36/TT OTL O:0.0/10 NXB XIC T4:36/DN BST OTU O:0.0/10 NXB OTU B3:0/5 NXB MOV 99 N7:6 BND BND EOR
%   N7:6  RECAP_SEQ  "Recap Sequencer" %
%   I:0.1/1  HORIZ_RIGHT_IN %
%   I:0.0/15  LIFT_DOWN_IN %
%   O:0.0/9  LEFT_CAPPER_DOWN  "Left Capper Down" %
%   T4:36  RECAP_STEP_13 %
%   O:0.0/10  EJECT_LEFT  "Eject Left" %
%   B3:0/5  RECAP_LEFT  "Recap Left Side, Then Reset" %

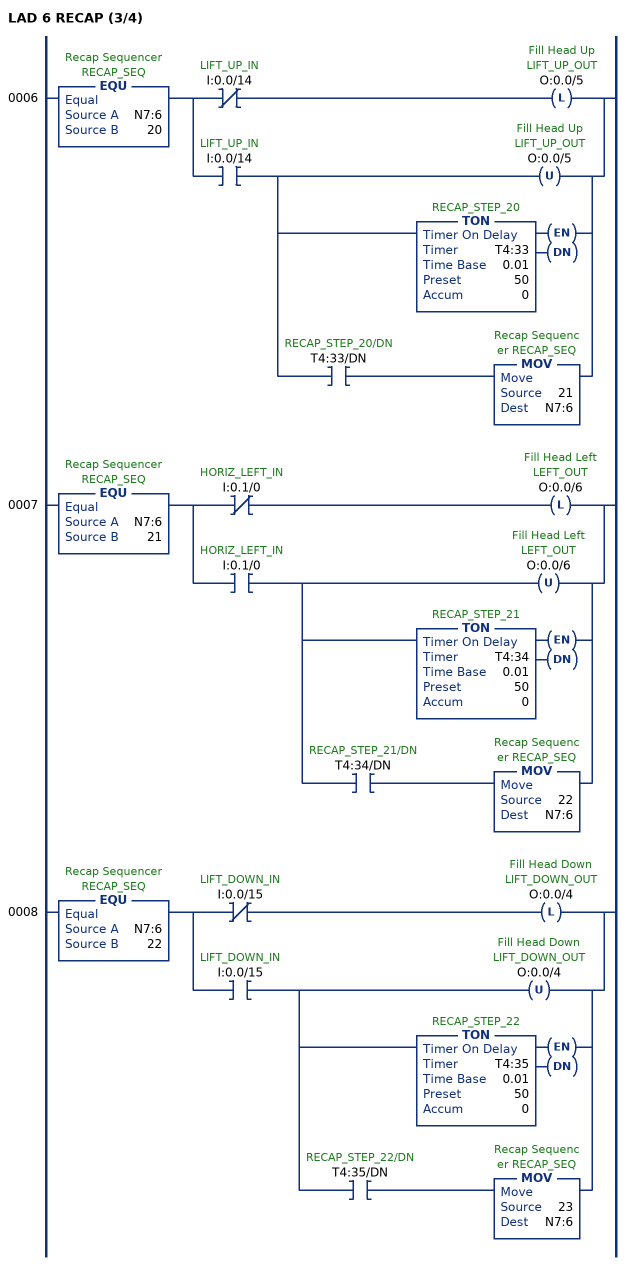
% Rung: 6 %
SOR EQU N7:6 20 BST XIO I:0.0/14 OTL O:0.0/5 NXB XIC I:0.0/14 BST OTU O:0.0/5 NXB TON T4:33 0.01 50 0 NXB XIC T4:33/DN MOV 21 N7:6 BND BND EOR
%   N7:6  RECAP_SEQ  "Recap Sequencer" %
%   I:0.0/14  LIFT_UP_IN %
%   O:0.0/5  LIFT_UP_OUT  "Fill Head Up" %
%   T4:33  RECAP_STEP_20 %
% Rung: 7 %
SOR EQU N7:6 21 BST XIO I:0.1/0 OTL O:0.0/6 NXB XIC I:0.1/0 BST OTU O:0.0/6 NXB TON T4:34 0.01 50 0 NXB XIC T4:34/DN MOV 22 N7:6 BND BND EOR
%   N7:6  RECAP_SEQ  "Recap Sequencer" %
%   I:0.1/0  HORIZ_LEFT_IN %
%   O:0.0/6  LEFT_OUT  "Fill Head Left" %
%   T4:34  RECAP_STEP_21 %
% Rung: 8 %
SOR EQU N7:6 22 BST XIO I:0.0/15 OTL O:0.0/4 NXB XIC I:0.0/15 BST OTU O:0.0/4 NXB TON T4:35 0.01 50 0 NXB XIC T4:35/DN MOV 23 N7:6 BND BND EOR
%   N7:6  RECAP_SEQ  "Recap Sequencer" %
%   I:0.0/15  LIFT_DOWN_IN %
%   O:0.0/4  LIFT_DOWN_OUT  "Fill Head Down" %
%   T4:35  RECAP_STEP_22 %

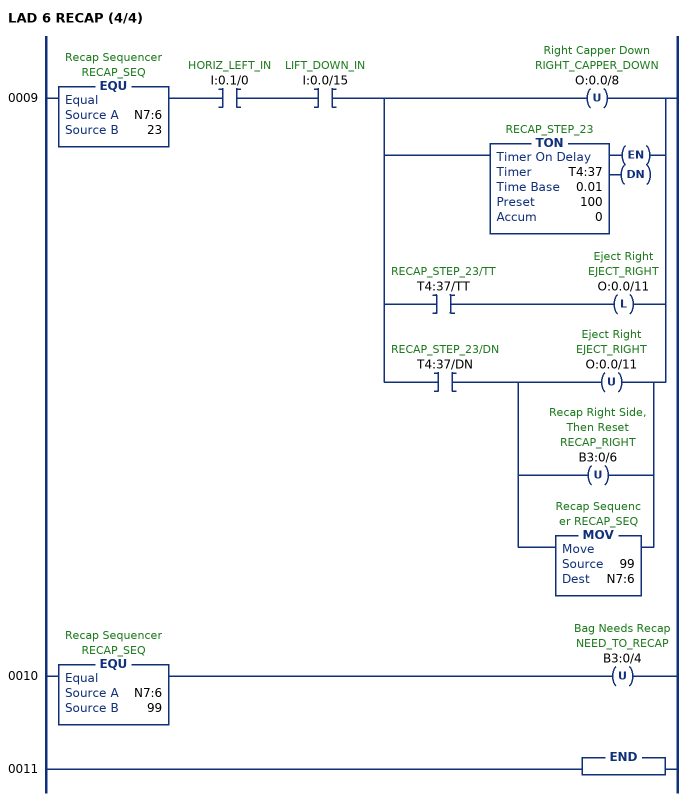
% Rung: 9 %
SOR EQU N7:6 23 XIC I:0.1/0 XIC I:0.0/15 BST OTU O:0.0/8 NXB TON T4:37 0.01 100 0 NXB XIC T4:37/TT OTL O:0.0/11 NXB XIC T4:37/DN BST OTU O:0.0/11 NXB OTU B3:0/6 NXB MOV 99 N7:6 BND BND EOR
%   N7:6  RECAP_SEQ  "Recap Sequencer" %
%   I:0.1/0  HORIZ_LEFT_IN %
%   I:0.0/15  LIFT_DOWN_IN %
%   O:0.0/8  RIGHT_CAPPER_DOWN  "Right Capper Down" %
%   T4:37  RECAP_STEP_23 %
%   O:0.0/11  EJECT_RIGHT  "Eject Right" %
%   B3:0/6  RECAP_RIGHT  "Recap Right Side, Then Reset" %
% Rung: 10 %
SOR EQU N7:6 99 OTU B3:0/4 EOR
%   N7:6  RECAP_SEQ  "Recap Sequencer" %
%   B3:0/4  NEED_TO_RECAP  "Bag Needs Recap" %
% Rung: 11 %
SOR END EOR

OTHER DOCUMENTED ADDRESSES
  B3:1/5  MAN_FILL_CLOSE  "Manuial Fill Valve Close"
  B3:1/6  MAN_LEFT_GATE_OPEN  "Manual Left Gate Open"
  B3:1/7  MAN_RIGHT_GATE_OPEN  "Manual Right Gate Open"
  B3:20  ONE_SHOTS
  DFILE:0  "OUTPUT"
  DFILE:1  "INPUT"
  DFILE:2  "STATUS"
  DFILE:3  "BINARY"
  DFILE:4  "TIMER"
  DFILE:5  "COUNTER"
  DFILE:6  "CONTROL"
  DFILE:7  "INTEGER"
  DFILE:8  "FLOAT"
  I:1.0/1  ABORT_BUTTON
  I:1.0/4  DOOR_SWITCH
  I:1.0/5  CANCEL_FILL_SWITCH
  I:2.0/7  FILL_COMPLETE
  T4:5  COUNT_RESET_DELAY
  T4:13  STEP_4_DELAY
  T4:15  STEP_7_DELAY

REVISION NOTES
  0: Reautomation October 2007

DATA TABLE (non-zero values as saved)
DATA B3
% B3:0 % 0X0008 0X0000 0X0000 0X0000 0X0000 0X0000 0X0000 0X0000 0X0000 0X0000
% B3:20 % 0X0030
DATA T4
% .PRE .ACC %
% T4:0 % 150 0
% T4:1 % 100 0
% T4:2 % 100 0
% T4:3 % 75 0
% T4:4 % 100 0
% T4:5 % 50 0
% T4:10 % 50 0
% T4:11 % 50 0
% T4:12 % 50 0
% T4:13 % 180 0
% T4:14 % 50 0
% T4:15 % 150 92
% T4:16 % 50 0
% T4:20 % 50 0
% T4:21 % 100 0
% T4:22 % 50 0
% T4:23 % 50 0
% T4:24 % 75 0
% T4:25 % 100 0
% T4:30 % 50 0
% T4:31 % 50 0
% T4:32 % 50 0
% T4:33 % 50 0
% T4:34 % 50 0
% T4:35 % 50 0
% T4:36 % 100 0
% T4:37 % 100 0
